// TwinCAT 3 PLC project plc
// ProgramVersion: 3.1.4024.0
// libraries:
//   Tc2_Standard, * (Beckhoff Automation GmbH)
//   Tc2_System, * (Beckhoff Automation GmbH)
//   Tc3_Module, * (Beckhoff Automation GmbH)
// project tree:
//   / PlcTask.TcTTO
//   POUs/ LLD.TcPOU, MAIN.TcPOU
// real-time tasks:
//   TASK PlcTask: cycle T#10ms, priority 20, ADS port 350

CONFIGURATION plc
    RESOURCE PLC ON TwinCAT3
        TASK PlcTask(INTERVAL := T#10ms, PRIORITY := 20);
        PROGRAM MAIN WITH PlcTask : MAIN;
    END_RESOURCE
END_CONFIGURATION

// ---- POUs/MAIN.TcPOU
PROGRAM MAIN
VAR
END_VAR

LLD();

END_PROGRAM

// ---- POUs/LLD.TcPOU
PROGRAM LLD
VAR
	i : INT := 0;
	f : REAL := 0.0;
	elapsed : TIME := TIME#0M0S0MS;
	today : DATE := DATE#2023-05-19;
	message : STRING := '';
	count : BYTE := 0;
	
	A AT %I* : BOOL := FALSE;
	B AT %I* : BOOL := FALSE;
	C AT %I* : BOOL := FALSE;
	D AT %Q* : BOOL := FALSE;
	
	op1 : INT := 1;
	op2 : INT := 2;
	res : REAL := 0.0;
	test : BOOL := FALSE;
	
	TON_0 : TON;
END_VAR

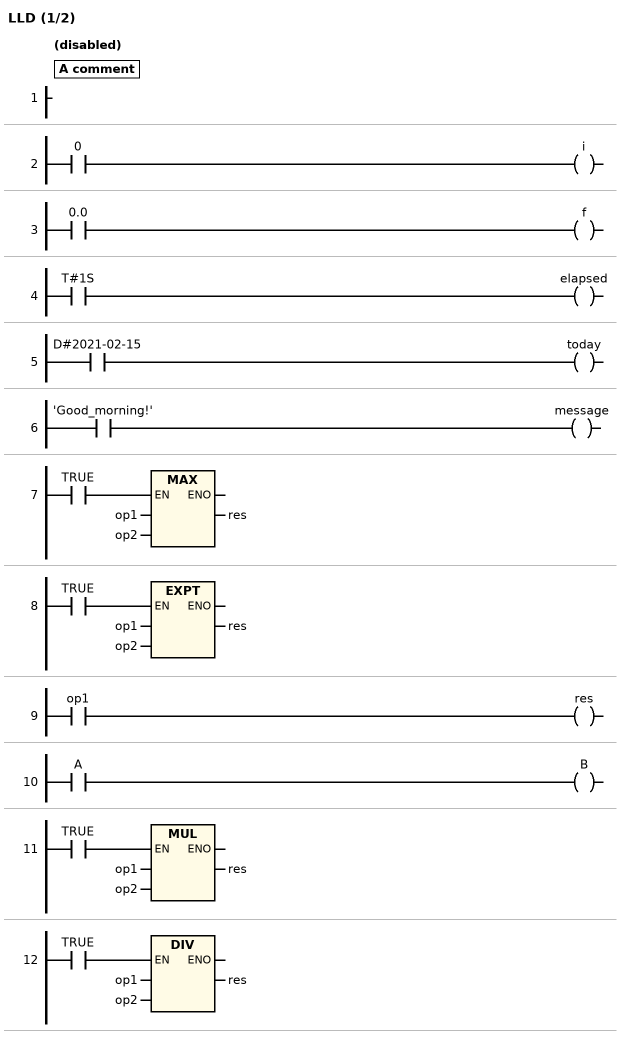
// NETWORK 1 (disabled)
// label: A comment

// NETWORK 2
i := 0;

// NETWORK 3
f := 0.0;

// NETWORK 4
elapsed := T#1S;

// NETWORK 5
today := D#2021-02-15;

// NETWORK 6
message := 'Good_morning!';

// NETWORK 7
res := MAX(op1, op2);

// NETWORK 8
res := EXPT(op1, op2);

// NETWORK 9
res := op1;

// NETWORK 10
B := A;

// NETWORK 11
res := op1 * op2;

// NETWORK 12
res := op1 / op2;

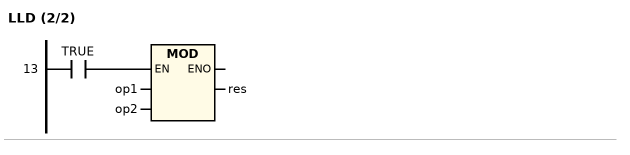
// NETWORK 13
res := op1 MOD op2;

END_PROGRAM
